// TIA Portal V20 export
TYPE "ScaVal"
   STRUCT
      High : Real := 100.0;   // High Value
      Low : Real;   // Low Value
   END_STRUCT;
END_TYPE
